(* Logix 5000 project; controller Evlog vendor 1 type 14 code 15 rev 20.11; software revision 20.05 *)

TASK MainTask (continuous, watchdog 500 ms) : MainProgram

MODULES
   Local : vendor 1 type 14 code 15 (SoftLogixController 2, rev 20.11)
      EIP : vendor 1 type 12 code 135 (SoftLogixVB 3, Ethernet 172.22.255.153, rev 20.1)
END_MODULES

TYPE STRING484 :
STRUCT
   LEN : DINT;
   DATA : SINT[480];
END_STRUCT
END_TYPE

TYPE u_EventTable :
STRUCT
   Ons_Short : BOOL[512];
   Last_Status : BOOL[1024];
END_STRUCT
END_TYPE

TYPE u_Timer :
STRUCT
   Yer : INT;
   Month : SINT;
   Day : SINT;
   Hour : SINT;
   Minute : SINT;
   Sec : SINT;
   MillSec : DINT;
END_STRUCT
END_TYPE

TYPE uEventsDB :
STRUCT
   Events : uEvlent[1024];
   NextEvent : INT;
   LastLostEvent : INT;
   EventOverFlow : BOOL;
   RemainderValidEvent : INT;
END_STRUCT
END_TYPE

TYPE uEvlent :   // @Ver 1.0
STRUCT
   ID : INT;   // Event ID
   Active : BOOL;
   IsSend : BOOL;
   Time : u_Timer;
END_STRUCT
END_TYPE

TYPE uSendMsg :   // @Ver 1.0
STRUCT
   MsgCount : SINT;
   BufferNotEmpty : BOOL;
   EmptyBuffer : uEvlent;
   SendBuffer : uEvlent;
   SendMSG : STRING;
END_STRUCT
END_TYPE

ADD_ON_INSTRUCTION CreateSendEvent   (* revision 1.0 *)
VAR_IN_OUT
   io_EvDB : uEventsDB; {required}
   o_SendBuffer : uSendMsg; {required}
END_VAR
VAR_INPUT
   Mutil_EvSend : BOOL; {access None, visible}
END_VAR
VAR_OUTPUT
   o_Error : BOOL; {access None}
END_VAR
VAR
   LocalEvDB : uEventsDB; {access None}
   True : BOOL; {access None}
   False : BOOL; {access None}
   i : DINT; {access None}
   Max_MsgCount : DINT; {access None}
   Last_index : DINT; {access None}
   MsgIndex : DINT; {access None}
   Temp_ID : STRING; {access None}
   Temp_Time : STRING; {access None}
   TIMEToSTRING : TIME_To_STRING; {access None}
   Index : DINT; {access None}
   Delimit : SINT; {access None}
   Split : STRING; {access None}
   Temp_Str : STRING; {access None}
   Time2Str : TIME_To_STRING; {access None}
   tempCount : DINT; {access None}
   EndOfCount : DINT; {access None}
   Tem_Str1 : STRING; {access None}
END_VAR

ROUTINE Logic   (* structured text *)
   
   True :=1;
   False:=0;
   Split.DATA[0]:=58;
   Split.Len:=1;
   Max_MsgCount:=500;
   o_Error:=False;
   Temp_Str.Len:=0;
   
   //
   
   IF Not o_SendBuffer.BufferNotEmpty Then
      o_SendBuffer.SendMSG.Len:=0;
   END_IF;
   
   //Mssage: ID:Timer:
   IF  io_EvDB.NextEvent>1 AND Not o_SendBuffer.BufferNotEmpty Then
       IF Not Mutil_EvSend then
   	   Cop(io_EvDB.Events[io_EvDB.NextEvent-1], o_SendBuffer.SendBuffer,1);
          //Cop(o_SendBuffer.EmptyBuffer, io_EvDB.Events[io_EvDB.NextEvent],1);
          DTOS(o_SendBuffer.SendBuffer.ID,Temp_Str);
   	   Concat(o_SendBuffer.SendMSG,Temp_Str,o_SendBuffer.SendMSG);
   	   Temp_Str.Len:=0;
          Concat(o_SendBuffer.SendMSG,Split,o_SendBuffer.SendMSG);
          TIME_To_STRING(Time2Str,o_SendBuffer.SendBuffer.Time,Temp_Str);
   	   Concat(o_SendBuffer.SendMSG,Temp_Str,o_SendBuffer.SendMSG);
          o_SendBuffer.BufferNotEmpty:=True;
          io_EvDB.NextEvent:=io_EvDB.NextEvent-1;
   	END_IF;
   
   END_IF;
   
   
   
   
   
   
   
   
   
   
   
   
   
   
   
   
   
   
   
   
   
   
   
   
   
   
   
   
   
   
   
   
   
   
   
   
   
   
   
   
   
   
   
   
   
   
   
END_ROUTINE
END_ADD_ON_INSTRUCTION

ADD_ON_INSTRUCTION CreatNewEvent   (* revision 1.0 *)
VAR_INPUT
   Enbale : DINT;
   Single_Input : BOOL; {required}
   Ev_ID : DINT; {access None, required}
END_VAR
VAR_IN_OUT
   IO_EvDB : uEventsDB; {required}
END_VAR
VAR_INPUT
   o_Parem_Err : BOOL; {access None, required}
END_VAR
VAR_IN_OUT
   Ev_Table : u_EventTable; {required}
END_VAR
VAR
   DT : DINT[6]; {access None}
   LocalIndex : DINT; {access None}
   Single_Trig : BOOL[1024]; {access None}
   OnsHelper : BOOL[1024]; {access None}
   Temp_SwitchSingle : BOOL; {access None}
   False : BOOL; {access None}
   True : BOOL; {access None}
   Max_ID : DINT; {access None}
   LocalDateTime : DINT[7]; {access None}
   Local_EvDB : uEvlent[1001]; {access None}
END_VAR

ROUTINE Logic   (* structured text *)
   
   (*
   VERSIONS:
   
   V1.0    |   Jerry  | First release
   
   
   1.单周期内  如果ID不一致 ,产生新的事件记录
   2.不同周期下,如果信号被重新触发,产生新的事件记录.
   3.同一事件,如果下一个周期没有产生上升沿 将不会记录.
   
   *)
   
   (*
   VERSION : '1.0'
   AUTHOR  : Jerry
   NAME    : EVENT
   FAMILY  : global
   *)
   
   True   :=1;
   False  :=0;
   Max_ID :=1000;//此处UDT 定义为1024
   
   Temp_SwitchSingle:=Single_Input;    //Cop  到本地 确保  本次程序结束能够复位状态,使下一次调用重新初始化
   IF Ev_ID>Max_ID OR Ev_ID<=0 Then
      o_Parem_Err:=True;
      Ev_ID:=1;
   END_IF;
   
   IF IO_EvDB.NextEvent>Max_ID OR IO_EvDB.NextEvent<=0 Then
      IO_EvDB.NextEvent:=1;
   END_IF;
   
   IF  Temp_SwitchSingle and not Ev_Table.Last_Status[Ev_ID] then
       Ev_Table.Last_Status[Ev_ID]:=True;
   //添加事件时间到Buffer
       GSV(WallClockTime,,DateTime,LocalDateTime[0]);
       IO_EvDB.Events[IO_EvDB.NextEvent].Time.Yer   :=LocalDateTime[0];
       IO_EvDB.Events[IO_EvDB.NextEvent].Time.Month :=LocalDateTime[1];
   	IO_EvDB.Events[IO_EvDB.NextEvent].Time.day   :=LocalDateTime[2];
   	IO_EvDB.Events[IO_EvDB.NextEvent].Time.hour  :=LocalDateTime[3];
   	IO_EvDB.Events[IO_EvDB.NextEvent].Time.minute:=LocalDateTime[4];
   	IO_EvDB.Events[IO_EvDB.NextEvent].Time.Sec   :=LocalDateTime[5];
   	IO_EvDB.Events[IO_EvDB.NextEvent].Time.MillSec:=LocalDateTime[6];
   
   	//添加事件ID到Buffer
   	IO_EvDB.Events[IO_EvDB.NextEvent].ID:=Ev_ID;
   	IO_EvDB.Events[IO_EvDB.NextEvent].Active:=True;
       IO_EvDB.Events[IO_EvDB.NextEvent].IsSend:=False;
   	IO_EvDB.NextEvent:=IO_EvDB.NextEvent+1;
   	IO_EvDB.RemainderValidEvent:=IO_EvDB.RemainderValidEvent+1;
   	IF IO_EvDB.NextEvent>Max_ID then
   	   IO_EvDB.NextEvent:=1;
          IO_EvDB.EventOverFlow:=True;
   	END_IF;
   End_IF;
   
   
   IF Not Temp_SwitchSingle and Ev_Table.Last_Status[Ev_ID] then
      Ev_Table.Last_Status[Ev_ID]:=False;
   END_IF;
   
   
   
   
   
END_ROUTINE
END_ADD_ON_INSTRUCTION

ADD_ON_INSTRUCTION CreatSendMsg   (* revision 1.0 *)
VAR_IN_OUT
   io_EvDB : uEventsDB; {required}
   o_SendMSG : uSendMsg; {required}
   Time2Str1 : TIME_To_STRING; {required}
END_VAR
VAR
   Split : STRING := ':'; {access None}
   Temp_Str : STRING; {access None}
   Time2Str : TIME_To_STRING; {access None}
END_VAR

ROUTINE Logic   (* ladder *)
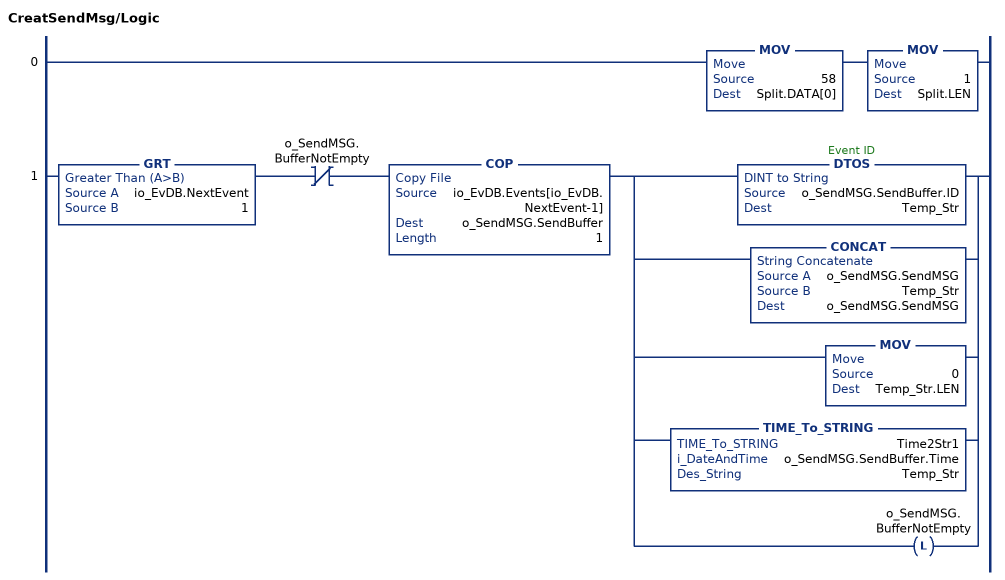
   0: MOV(58,Split.DATA[0])MOV(1,Split.LEN);
   1: GRT(io_EvDB.NextEvent,1)XIO(o_SendMSG.BufferNotEmpty)COP(io_EvDB.Events[io_EvDB.NextEvent-1],o_SendMSG.SendBuffer,1)[DTOS(o_SendMSG.SendBuffer.ID,Temp_Str) ,CONCAT(o_SendMSG.SendMSG,Temp_Str,o_SendMSG.SendMSG) ,MOV(0,Temp_Str.LEN) ,TIME_To_STRING(Time2Str1,o_SendMSG.SendBuffer.Time,Temp_Str) ,OTL(o_SendMSG.BufferNotEmpty) ];
END_ROUTINE
END_ADD_ON_INSTRUCTION

ADD_ON_INSTRUCTION TIME_To_STRING   (* revision 1.0 *)
VAR_IN_OUT
   i_DateAndTime : u_Timer; {required}
   Des_String : STRING; {required}
END_VAR
VAR
   i : DINT; {access None}
   Temp_Str : STRING; {access None}
   Split : STRING := '.'; {access None}
END_VAR

ROUTINE Logic   (* structured text *)
   
   
   Des_String.len:=0;
         DTOS(i_DateAndTime.Yer,Temp_Str);
      Concat(Des_String,Temp_Str,Des_String);
      Concat(Des_String,Split,Des_String);
      Temp_Str.Len:=0;
         DTOS(i_DateAndTime.Month,Temp_Str);
      Concat(Des_String,Temp_Str,Des_String);
      Concat(Des_String,Split,Des_String);
      Temp_Str.Len:=0;
         DTOS(i_DateAndTime.Day,Temp_Str);
      Concat(Des_String,Temp_Str,Des_String);
      Concat(Des_String,Split,Des_String);
      Temp_Str.Len:=0;
         DTOS(i_DateAndTime.Hour,Temp_Str);
      Concat(Des_String,Temp_Str,Des_String);
      Concat(Des_String,Split,Des_String);
      Temp_Str.Len:=0;
         DTOS(i_DateAndTime.Minute,Temp_Str);
      Concat(Des_String,Temp_Str,Des_String);
      Concat(Des_String,Split,Des_String);
      Temp_Str.Len:=0;
          DTOS(i_DateAndTime.Sec,Temp_Str);
      Concat(Des_String,Temp_Str,Des_String);
      Concat(Des_String,Split,Des_String);
   Temp_Str.Len:=0;
          DTOS(i_DateAndTime.MillSec,Temp_Str);
      Concat(Des_String,Temp_Str,Des_String);
END_ROUTINE
END_ADD_ON_INSTRUCTION

VAR_GLOBAL   (* controller tags *)
   booltest : BOOL := 1;
   Ev_Table : u_EventTable;
   EvMsgDB : uEvlent[10000];
   SendBuffer : uSendMsg := (MsgCount := 1, SendBuffer.ID := 1, SendBuffer.Active := 1, SendBuffer.Time.Yer := 2022, SendBuffer.Time.Month := 2, SendBuffer.Time.Day := 5, SendBuffer.Time.Hour := 14, SendBuffer.Time.Minute := 40, SendBuffer.Time.Sec := 40, SendBuffer.Time.MillSec := 175138);
   SendMsg_Buffer : uSendMsg := (BufferNotEmpty := 1);
   string1 : STRING := '123456';
   test : BOOL;
   testStr : STRING;
   Time2Str : TIME_To_STRING;
END_VAR

PROGRAM MainProgram   (* main routine MainRoutine *)
VAR
   CreatMSG : CreatSendMsg;
   ddd : DINT := 2022;
   Ev_Table : u_EventTable := (Last_Status[1] := 1);
   EvDB : uEvlent[1000] := ([0].ID := 1, [0].Active := 1, [1].ID := 2, [1].Active := 1, [2].ID := 1, [2].Active := 1, [3].ID := 2, [3].Active := 1, [4].ID := 1, [4].Active := 1, [5].ID := 2, [5].Active := 1, [6].ID := 1, [6].Active := 1, [7].ID := 2, [7].Active := 1, [8].ID := 1, [8].Active := 1, [9].ID := 2, [9].Active := 1, [10].ID := 1, [10].Active := 1, [11].ID := 2, [11].Active := 1, [12].ID := 1, [12].Active := 1, [13].ID := 2, [13].Active := 1, [14].ID := 1, [14].Active := 1, [15].ID := 2, [15].Active := 1, [16].ID := 1, [16].Active := 1, [17].ID := 2, [17].Active := 1, [18].ID := 1, [18].Active := 1, [19].ID := 2, [19].Active := 1, [20].ID := 1, [20].Active := 1, [21].ID := 2, [21].Active := 1, [22].ID := 1, [22].Active := 1, [23].ID := 2, [23].Active := 1, [24].ID := 1, [24].Active := 1, [25].ID := 2, [25].Active := 1, [26].ID := 1, [26].Active := 1, [27].ID := 2, [27].Active := 1, [28].ID := 1, [28].Active := 1, [29].ID := 2, [29].Active := 1,
        [30].ID := 1, [30].Active := 1, [31].ID := 2, [31].Active := 1, [32].ID := 1, [32].Active := 1, [33].ID := 2, [33].Active := 1, [34].ID := 1, [34].Active := 1, [35].ID := 2, [35].Active := 1, [36].ID := 1, [36].Active := 1, [37].ID := 2, [37].Active := 1, [38].ID := 1, [38].Active := 1, [39].ID := 2, [39].Active := 1, [40].ID := 1, [40].Active := 1, [41].ID := 2, [41].Active := 1, [42].ID := 1, [42].Active := 1, [43].ID := 2, [43].Active := 1, [44].ID := 1, [44].Active := 1, [45].ID := 2, [45].Active := 1, [46].ID := 1, [46].Active := 1, [47].ID := 2, [47].Active := 1, [48].ID := 1, [48].Active := 1, [49].ID := 2, [49].Active := 1, [50].ID := 1, [50].Active := 1, [51].ID := 2, [51].Active := 1, [52].ID := 1, [52].Active := 1, [53].ID := 2, [53].Active := 1, [54].ID := 1, [54].Active := 1, [55].ID := 2, [55].Active := 1, [56].ID := 1, [56].Active := 1, [57].ID := 2, [57].Active := 1, [58].ID := 1, [58].Active := 1, [59].ID := 2, [59].Active := 1,
        [60].ID := 1, [60].Active := 1, [61].ID := 2, [61].Active := 1, [62].ID := 1, [62].Active := 1, [63].ID := 2, [63].Active := 1, [64].ID := 1, [64].Active := 1, [65].ID := 2, [65].Active := 1, [66].ID := 1, [66].Active := 1, [67].ID := 2, [67].Active := 1, [68].ID := 1, [68].Active := 1, [69].ID := 2, [69].Active := 1, [70].ID := 1, [70].Active := 1, [71].ID := 2, [71].Active := 1, [72].ID := 1, [72].Active := 1, [73].ID := 2, [73].Active := 1, [74].ID := 1, [74].Active := 1, [75].ID := 2, [75].Active := 1, [76].ID := 1, [76].Active := 1, [77].ID := 2, [77].Active := 1, [78].ID := 1, [78].Active := 1, [79].ID := 2, [79].Active := 1, [80].ID := 1, [80].Active := 1, [81].ID := 2, [81].Active := 1, [82].ID := 1, [82].Active := 1, [83].ID := 2, [83].Active := 1, [84].ID := 1, [84].Active := 1, [85].ID := 2, [85].Active := 1, [86].ID := 1, [86].Active := 1, [87].ID := 2, [87].Active := 1, [88].ID := 1, [88].Active := 1, [89].ID := 2, [89].Active := 1,
        [90].ID := 1, [90].Active := 1, [91].ID := 2, [91].Active := 1, [92].ID := 1, [92].Active := 1, [93].ID := 2, [93].Active := 1, [94].ID := 1, [94].Active := 1, [95].ID := 2, [95].Active := 1, [96].ID := 1, [96].Active := 1, [97].ID := 2, [97].Active := 1, [98].ID := 1, [98].Active := 1, [99].ID := 2, [99].Active := 1, [100].ID := 1, [100].Active := 1, [101].ID := 2, [101].Active := 1, [102].ID := 1, [102].Active := 1, [103].ID := 2, [103].Active := 1, [104].ID := 1, [104].Active := 1, [105].ID := 2, [105].Active := 1, [106].ID := 1, [106].Active := 1, [107].ID := 2, [107].Active := 1, [108].ID := 1, [108].Active := 1, [109].ID := 2, [109].Active := 1, [110].ID := 1, [110].Active := 1, [111].ID := 2, [111].Active := 1, [112].ID := 1, [112].Active := 1, [113].ID := 2, [113].Active := 1, [114].ID := 1, [114].Active := 1, [115].ID := 2, [115].Active := 1, [116].ID := 1, [116].Active := 1, [117].ID := 2, [117].Active := 1, [118].ID := 1, [118].Active := 1, [119].ID := 2, [119].Active := 1,
        [120].ID := 1, [120].Active := 1, [121].ID := 2, [121].Active := 1, [122].ID := 1, [122].Active := 1, [123].ID := 2, [123].Active := 1, [124].ID := 1, [124].Active := 1, [125].ID := 2, [125].Active := 1, [126].ID := 1, [126].Active := 1, [127].ID := 2, [127].Active := 1, [128].ID := 1, [128].Active := 1, [129].ID := 2, [129].Active := 1, [130].ID := 1, [130].Active := 1, [131].ID := 2, [131].Active := 1, [132].ID := 1, [132].Active := 1, [133].ID := 2, [133].Active := 1, [134].ID := 1, [134].Active := 1, [135].ID := 2, [135].Active := 1, [136].ID := 1, [136].Active := 1, [137].ID := 2, [137].Active := 1, [138].ID := 1, [138].Active := 1, [139].ID := 2, [139].Active := 1, [140].ID := 1, [140].Active := 1, [141].ID := 2, [141].Active := 1, [142].ID := 1, [142].Active := 1, [143].ID := 2, [143].Active := 1, [144].ID := 1, [144].Active := 1, [145].ID := 2, [145].Active := 1, [146].ID := 1, [146].Active := 1, [147].ID := 2, [147].Active := 1, [148].ID := 1, [148].Active := 1, [149].ID := 2, [149].Active := 1,
        [150].ID := 1, [150].Active := 1, [151].ID := 2, [151].Active := 1, [152].ID := 1, [152].Active := 1, [153].ID := 2, [153].Active := 1, [154].ID := 1, [154].Active := 1, [155].ID := 2, [155].Active := 1, [156].ID := 1, [156].Active := 1, [157].ID := 2, [157].Active := 1, [158].ID := 1, [158].Active := 1, [159].ID := 2, [159].Active := 1, [160].ID := 1, [160].Active := 1, [161].ID := 2, [161].Active := 1, [162].ID := 1, [162].Active := 1, [163].ID := 2, [163].Active := 1, [164].ID := 1, [164].Active := 1, [165].ID := 2, [165].Active := 1, [166].ID := 1, [166].Active := 1, [167].ID := 2, [167].Active := 1, [168].ID := 1, [168].Active := 1, [169].ID := 2, [169].Active := 1, [170].ID := 1, [170].Active := 1, [171].ID := 2, [171].Active := 1, [172].ID := 2, [172].Active := 1, [173].ID := 1, [173].Active := 1, [174].ID := 2, [174].Active := 1, [175].ID := 1, [175].Active := 1, [176].ID := 2, [176].Active := 1, [177].ID := 1, [177].Active := 1, [178].ID := 2, [178].Active := 1, [179].ID := 1, [179].Active := 1,
        [180].ID := 2, [180].Active := 1, [181].ID := 1, [181].Active := 1, [182].ID := 2, [182].Active := 1, [183].ID := 1, [183].Active := 1, [184].ID := 2, [184].Active := 1, [185].ID := 1, [185].Active := 1, [186].ID := 2, [186].Active := 1, [187].ID := 1, [187].Active := 1, [188].ID := 2, [188].Active := 1, [189].ID := 1, [189].Active := 1, [190].ID := 2, [190].Active := 1, [191].ID := 1, [191].Active := 1, [192].ID := 2, [192].Active := 1, [193].ID := 1, [193].Active := 1, [194].ID := 2, [194].Active := 1, [195].ID := 1, [195].Active := 1, [196].ID := 2, [196].Active := 1, [197].ID := 1, [197].Active := 1, [198].ID := 2, [198].Active := 1, [199].ID := 1, [199].Active := 1, [200].ID := 2, [200].Active := 1, [201].ID := 1, [201].Active := 1, [202].ID := 2, [202].Active := 1, [203].ID := 1, [203].Active := 1, [204].ID := 2, [204].Active := 1, [205].ID := 1, [205].Active := 1, [206].ID := 2, [206].Active := 1, [207].ID := 1, [207].Active := 1, [208].ID := 2, [208].Active := 1, [209].ID := 1, [209].Active := 1,
        [210].ID := 2, [210].Active := 1, [211].ID := 1, [211].Active := 1, [212].ID := 2, [212].Active := 1, [213].ID := 1, [213].Active := 1, [214].ID := 2, [214].Active := 1, [215].ID := 1, [215].Active := 1, [216].ID := 2, [216].Active := 1, [217].ID := 1, [217].Active := 1, [218].ID := 2, [218].Active := 1, [219].ID := 1, [219].Active := 1, [220].ID := 2, [220].Active := 1, [221].ID := 1, [221].Active := 1, [222].ID := 2, [222].Active := 1, [223].ID := 1, [223].Active := 1, [224].ID := 2, [224].Active := 1, [225].ID := 1, [225].Active := 1, [226].ID := 2, [226].Active := 1, [227].ID := 1, [227].Active := 1, [228].ID := 2, [228].Active := 1, [229].ID := 1, [229].Active := 1, [230].ID := 2, [230].Active := 1, [231].ID := 1, [231].Active := 1, [232].ID := 2, [232].Active := 1, [233].ID := 1, [233].Active := 1, [234].ID := 2, [234].Active := 1, [235].ID := 1, [235].Active := 1, [236].ID := 2, [236].Active := 1, [237].ID := 1, [237].Active := 1, [238].ID := 2, [238].Active := 1, [239].ID := 1, [239].Active := 1,
        [240].ID := 2, [240].Active := 1, [241].ID := 1, [241].Active := 1, [242].ID := 2, [242].Active := 1, [243].ID := 1, [243].Active := 1, [244].ID := 2, [244].Active := 1, [245].ID := 1, [245].Active := 1, [246].ID := 2, [246].Active := 1, [247].ID := 1, [247].Active := 1, [248].ID := 2, [248].Active := 1, [249].ID := 1, [249].Active := 1, [250].ID := 2, [250].Active := 1, [251].ID := 1, [251].Active := 1, [252].ID := 2, [252].Active := 1, [253].ID := 1, [253].Active := 1, [254].ID := 2, [254].Active := 1, [255].ID := 1, [255].Active := 1, [256].ID := 2, [256].Active := 1, [257].ID := 1, [257].Active := 1, [258].ID := 2, [258].Active := 1, [259].ID := 1, [259].Active := 1, [260].ID := 2, [260].Active := 1, [261].ID := 1, [261].Active := 1, [262].ID := 2, [262].Active := 1, [263].ID := 1, [263].Active := 1, [264].ID := 2, [264].Active := 1, [265].ID := 1, [265].Active := 1, [266].ID := 2, [266].Active := 1, [267].ID := 1, [267].Active := 1, [268].ID := 2, [268].Active := 1, [269].ID := 1, [269].Active := 1,
        [270].ID := 2, [270].Active := 1, [271].ID := 1, [271].Active := 1, [272].ID := 2, [272].Active := 1, [273].ID := 1, [273].Active := 1, [274].ID := 2, [274].Active := 1, [275].ID := 1, [275].Active := 1, [276].ID := 2, [276].Active := 1, [277].ID := 1, [277].Active := 1, [278].ID := 2, [278].Active := 1, [279].ID := 1, [279].Active := 1, [280].ID := 2, [280].Active := 1, [281].ID := 1, [281].Active := 1, [282].ID := 2, [282].Active := 1, [283].ID := 1, [283].Active := 1, [284].ID := 2, [284].Active := 1, [285].ID := 1, [285].Active := 1, [286].ID := 2, [286].Active := 1, [287].ID := 1, [287].Active := 1, [288].ID := 2, [288].Active := 1, [289].ID := 1, [289].Active := 1, [290].ID := 2, [290].Active := 1, [291].ID := 1, [291].Active := 1, [292].ID := 2, [292].Active := 1, [293].ID := 1, [293].Active := 1, [294].ID := 2, [294].Active := 1, [295].ID := 1, [295].Active := 1, [296].ID := 2, [296].Active := 1, [297].ID := 1, [297].Active := 1, [298].ID := 2, [298].Active := 1, [299].ID := 1, [299].Active := 1,
        [300].ID := 2, [300].Active := 1, [301].ID := 1, [301].Active := 1, [302].ID := 2, [302].Active := 1, [303].ID := 1, [303].Active := 1, [304].ID := 2, [304].Active := 1, [305].ID := 1, [305].Active := 1, [306].ID := 2, [306].Active := 1, [307].ID := 1, [307].Active := 1, [308].ID := 2, [308].Active := 1, [309].ID := 1, [309].Active := 1, [310].ID := 2, [310].Active := 1, [311].ID := 1, [311].Active := 1, [312].ID := 2, [312].Active := 1, [313].ID := 1, [313].Active := 1, [314].ID := 2, [314].Active := 1, [315].ID := 1, [315].Active := 1, [316].ID := 2, [316].Active := 1, [317].ID := 1, [317].Active := 1, [318].ID := 2, [318].Active := 1, [319].ID := 1, [319].Active := 1, [320].ID := 2, [320].Active := 1, [321].ID := 1, [321].Active := 1, [322].ID := 2, [322].Active := 1, [323].ID := 1, [323].Active := 1, [324].ID := 2, [324].Active := 1, [325].ID := 1, [325].Active := 1, [326].ID := 2, [326].Active := 1, [327].ID := 1, [327].Active := 1, [328].ID := 2, [328].Active := 1, [329].ID := 1, [329].Active := 1,
        [330].ID := 2, [330].Active := 1, [331].ID := 1, [331].Active := 1, [332].ID := 2, [332].Active := 1, [333].ID := 1, [333].Active := 1, [334].ID := 2, [334].Active := 1, [335].ID := 1, [335].Active := 1, [336].ID := 2, [336].Active := 1, [337].ID := 1, [337].Active := 1, [338].ID := 2, [338].Active := 1, [339].ID := 1, [339].Active := 1, [340].ID := 2, [340].Active := 1, [341].ID := 1, [341].Active := 1, [342].ID := 2, [342].Active := 1, [343].ID := 1, [343].Active := 1, [344].ID := 2, [344].Active := 1, [345].ID := 1, [345].Active := 1, [346].ID := 2, [346].Active := 1, [347].ID := 1, [347].Active := 1, [348].ID := 2, [348].Active := 1, [349].ID := 1, [349].Active := 1, [350].ID := 2, [350].Active := 1, [351].ID := 1, [351].Active := 1, [352].ID := 2, [352].Active := 1, [353].ID := 1, [353].Active := 1, [354].ID := 2, [354].Active := 1, [355].ID := 1, [355].Active := 1, [356].ID := 2, [356].Active := 1, [357].ID := 1, [357].Active := 1, [358].ID := 2, [358].Active := 1, [359].ID := 1, [359].Active := 1,
        [360].ID := 2, [360].Active := 1, [361].ID := 1, [361].Active := 1, [362].ID := 2, [362].Active := 1, [363].ID := 1, [363].Active := 1, [364].ID := 2, [364].Active := 1, [365].ID := 1, [365].Active := 1, [366].ID := 2, [366].Active := 1, [367].ID := 1, [367].Active := 1, [368].ID := 2, [368].Active := 1, [369].ID := 1, [369].Active := 1, [370].ID := 2, [370].Active := 1, [371].ID := 1, [371].Active := 1, [372].ID := 2, [372].Active := 1, [373].ID := 1, [373].Active := 1, [374].ID := 2, [374].Active := 1, [375].ID := 1, [375].Active := 1, [376].ID := 2, [376].Active := 1, [377].ID := 1, [377].Active := 1, [378].ID := 2, [378].Active := 1, [379].ID := 1, [379].Active := 1, [380].ID := 2, [380].Active := 1, [381].ID := 1, [381].Active := 1, [382].ID := 2, [382].Active := 1, [383].ID := 1, [383].Active := 1, [384].ID := 2, [384].Active := 1, [385].ID := 1, [385].Active := 1, [386].ID := 2, [386].Active := 1, [387].ID := 1, [387].Active := 1, [388].ID := 2, [388].Active := 1, [389].ID := 1, [389].Active := 1,
        [390].ID := 2, [390].Active := 1, [391].ID := 1, [391].Active := 1, [392].ID := 2, [392].Active := 1, [393].ID := 1, [393].Active := 1, [394].ID := 2, [394].Active := 1, [395].ID := 1, [395].Active := 1, [396].ID := 2, [396].Active := 1, [397].ID := 1, [397].Active := 1, [398].ID := 2, [398].Active := 1, [399].ID := 1, [399].Active := 1, [400].ID := 2, [400].Active := 1, [401].ID := 1, [401].Active := 1, [402].ID := 2, [402].Active := 1, [403].ID := 1, [403].Active := 1, [404].ID := 2, [404].Active := 1, [405].ID := 1, [405].Active := 1, [406].ID := 2, [406].Active := 1, [407].ID := 1, [407].Active := 1, [408].ID := 2, [408].Active := 1, [409].ID := 1, [409].Active := 1, [410].ID := 2, [410].Active := 1, [411].ID := 1, [411].Active := 1, [412].ID := 2, [412].Active := 1, [413].ID := 1, [413].Active := 1, [414].ID := 2, [414].Active := 1, [415].ID := 1, [415].Active := 1, [416].ID := 2, [416].Active := 1, [417].ID := 1, [417].Active := 1, [418].ID := 2, [418].Active := 1, [419].ID := 1, [419].Active := 1,
        [420].ID := 2, [420].Active := 1, [421].ID := 1, [421].Active := 1, [422].ID := 2, [422].Active := 1, [423].ID := 1, [423].Active := 1, [424].ID := 2, [424].Active := 1, [425].ID := 1, [425].Active := 1, [426].ID := 2, [426].Active := 1, [427].ID := 1, [427].Active := 1, [428].ID := 2, [428].Active := 1, [429].ID := 1, [429].Active := 1, [430].ID := 2, [430].Active := 1, [431].ID := 1, [431].Active := 1, [432].ID := 2, [432].Active := 1, [433].ID := 1, [433].Active := 1, [434].ID := 2, [434].Active := 1, [435].ID := 1, [435].Active := 1, [436].ID := 2, [436].Active := 1, [437].ID := 1, [437].Active := 1, [438].ID := 2, [438].Active := 1, [439].ID := 1, [439].Active := 1, [440].ID := 2, [440].Active := 1, [441].ID := 1, [441].Active := 1, [442].ID := 2, [442].Active := 1, [443].ID := 1, [443].Active := 1, [444].ID := 2, [444].Active := 1, [445].ID := 1, [445].Active := 1, [446].ID := 2, [446].Active := 1, [447].ID := 1, [447].Active := 1, [448].ID := 2, [448].Active := 1, [449].ID := 1, [449].Active := 1,
        [450].ID := 2, [450].Active := 1, [451].ID := 1, [451].Active := 1, [452].ID := 2, [452].Active := 1, [453].ID := 1, [453].Active := 1, [454].ID := 2, [454].Active := 1, [455].ID := 1, [455].Active := 1, [456].ID := 2, [456].Active := 1, [457].ID := 1, [457].Active := 1, [458].ID := 2, [458].Active := 1, [459].ID := 1, [459].Active := 1, [460].ID := 2, [460].Active := 1, [461].ID := 1, [461].Active := 1, [462].ID := 2, [462].Active := 1, [463].ID := 1, [463].Active := 1, [464].ID := 2, [464].Active := 1, [465].ID := 1, [465].Active := 1, [466].ID := 2, [466].Active := 1, [467].ID := 1, [467].Active := 1, [468].ID := 2, [468].Active := 1, [469].ID := 1, [469].Active := 1, [470].ID := 2, [470].Active := 1, [471].ID := 1, [471].Active := 1, [472].ID := 2, [472].Active := 1, [473].ID := 1, [473].Active := 1, [474].ID := 2, [474].Active := 1, [475].ID := 1, [475].Active := 1, [476].ID := 2, [476].Active := 1, [477].ID := 1, [477].Active := 1, [478].ID := 2, [478].Active := 1, [479].ID := 1, [479].Active := 1,
        [480].ID := 2, [480].Active := 1, [481].ID := 1, [481].Active := 1, [482].ID := 2, [482].Active := 1, [483].ID := 1, [483].Active := 1, [484].ID := 2, [484].Active := 1, [485].ID := 1, [485].Active := 1, [486].ID := 2, [486].Active := 1, [487].ID := 1, [487].Active := 1, [488].ID := 2, [488].Active := 1, [489].ID := 1, [489].Active := 1, [490].ID := 2, [490].Active := 1, [491].ID := 1, [491].Active := 1, [492].ID := 2, [492].Active := 1, [493].ID := 1, [493].Active := 1, [494].ID := 2, [494].Active := 1, [495].ID := 1, [495].Active := 1, [496].ID := 2, [496].Active := 1, [497].ID := 1, [497].Active := 1, [498].ID := 2, [498].Active := 1, [499].ID := 1, [499].Active := 1, [500].ID := 2, [500].Active := 1, [501].ID := 1, [501].Active := 1, [502].ID := 2, [502].Active := 1, [503].ID := 1, [503].Active := 1, [504].ID := 2, [504].Active := 1, [505].ID := 1, [505].Active := 1, [506].ID := 2, [506].Active := 1, [507].ID := 1, [507].Active := 1, [508].ID := 2, [508].Active := 1, [509].ID := 1, [509].Active := 1,
        [510].ID := 2, [510].Active := 1, [511].ID := 1, [511].Active := 1, [512].ID := 2, [512].Active := 1, [513].ID := 1, [513].Active := 1, [514].ID := 2, [514].Active := 1, [515].ID := 1, [515].Active := 1, [516].ID := 2, [516].Active := 1, [517].ID := 1, [517].Active := 1, [518].ID := 2, [518].Active := 1, [519].ID := 1, [519].Active := 1, [520].ID := 2, [520].Active := 1, [521].ID := 1, [521].Active := 1, [522].ID := 2, [522].Active := 1, [523].ID := 1, [523].Active := 1, [524].ID := 2, [524].Active := 1, [525].ID := 1, [525].Active := 1, [526].ID := 2, [526].Active := 1, [527].ID := 1, [527].Active := 1, [528].ID := 2, [528].Active := 1, [529].ID := 1, [529].Active := 1, [530].ID := 2, [530].Active := 1, [531].ID := 1, [531].Active := 1, [532].ID := 2, [532].Active := 1, [533].ID := 1, [533].Active := 1, [534].ID := 2, [534].Active := 1, [535].ID := 1, [535].Active := 1, [536].ID := 2, [536].Active := 1, [537].ID := 1, [537].Active := 1, [538].ID := 2, [538].Active := 1, [539].ID := 1, [539].Active := 1,
        [540].ID := 2, [540].Active := 1, [541].ID := 1, [541].Active := 1, [542].ID := 2, [542].Active := 1, [543].ID := 1, [543].Active := 1, [544].ID := 2, [544].Active := 1, [545].ID := 1, [545].Active := 1, [546].ID := 2, [546].Active := 1, [547].ID := 1, [547].Active := 1, [548].ID := 2, [548].Active := 1, [549].ID := 1, [549].Active := 1, [550].ID := 2, [550].Active := 1, [551].ID := 1, [551].Active := 1, [552].ID := 2, [552].Active := 1, [553].ID := 1, [553].Active := 1, [554].ID := 2, [554].Active := 1, [555].ID := 1, [555].Active := 1, [556].ID := 2, [556].Active := 1, [557].ID := 1, [557].Active := 1, [558].ID := 2, [558].Active := 1, [559].ID := 1, [559].Active := 1, [560].ID := 2, [560].Active := 1, [561].ID := 1, [561].Active := 1, [562].ID := 2, [562].Active := 1, [563].ID := 1, [563].Active := 1, [564].ID := 2, [564].Active := 1, [565].ID := 1, [565].Active := 1, [566].ID := 2, [566].Active := 1, [567].ID := 1, [567].Active := 1, [568].ID := 2, [568].Active := 1, [569].ID := 1, [569].Active := 1,
        [570].ID := 2, [570].Active := 1, [571].ID := 1, [571].Active := 1, [572].ID := 2, [572].Active := 1, [573].ID := 1, [573].Active := 1, [574].ID := 2, [574].Active := 1, [575].ID := 1, [575].Active := 1, [576].ID := 2, [576].Active := 1, [577].ID := 1, [577].Active := 1, [578].ID := 2, [578].Active := 1, [579].ID := 1, [579].Active := 1, [580].ID := 2, [580].Active := 1, [581].ID := 1, [581].Active := 1, [582].ID := 2, [582].Active := 1, [583].ID := 1, [583].Active := 1, [584].ID := 2, [584].Active := 1, [585].ID := 1, [585].Active := 1, [586].ID := 2, [586].Active := 1, [587].ID := 1, [587].Active := 1, [588].ID := 2, [588].Active := 1, [589].ID := 1, [589].Active := 1, [590].ID := 2, [590].Active := 1, [591].ID := 1, [591].Active := 1, [592].ID := 2, [592].Active := 1, [593].ID := 1, [593].Active := 1, [594].ID := 2, [594].Active := 1, [595].ID := 1, [595].Active := 1, [596].ID := 2, [596].Active := 1, [597].ID := 1, [597].Active := 1, [598].ID := 2, [598].Active := 1, [599].ID := 1, [599].Active := 1,
        [600].ID := 2, [600].Active := 1, [601].ID := 1, [601].Active := 1, [602].ID := 2, [602].Active := 1, [603].ID := 1, [603].Active := 1, [604].ID := 2, [604].Active := 1, [605].ID := 1, [605].Active := 1, [606].ID := 2, [606].Active := 1, [607].ID := 1, [607].Active := 1, [608].ID := 2, [608].Active := 1, [609].ID := 1, [609].Active := 1, [610].ID := 2, [610].Active := 1, [611].ID := 1, [611].Active := 1, [612].ID := 2, [612].Active := 1, [613].ID := 1, [613].Active := 1, [614].ID := 2, [614].Active := 1, [615].ID := 1, [615].Active := 1, [616].ID := 2, [616].Active := 1, [617].ID := 1, [617].Active := 1, [618].ID := 2, [618].Active := 1, [619].ID := 1, [619].Active := 1, [620].ID := 2, [620].Active := 1, [621].ID := 1, [621].Active := 1, [622].ID := 2, [622].Active := 1, [623].ID := 1, [623].Active := 1, [624].ID := 2, [624].Active := 1, [625].ID := 1, [625].Active := 1, [626].ID := 2, [626].Active := 1, [627].ID := 1, [627].Active := 1, [628].ID := 2, [628].Active := 1, [629].ID := 1, [629].Active := 1,
        [630].ID := 2, [630].Active := 1, [631].ID := 1, [631].Active := 1, [632].ID := 2, [632].Active := 1, [633].ID := 1, [633].Active := 1, [634].ID := 2, [634].Active := 1, [635].ID := 1, [635].Active := 1, [636].ID := 2, [636].Active := 1, [637].ID := 1, [637].Active := 1, [638].ID := 2, [638].Active := 1, [639].ID := 1, [639].Active := 1, [640].ID := 2, [640].Active := 1, [641].ID := 1, [641].Active := 1, [642].ID := 2, [642].Active := 1, [643].ID := 1, [643].Active := 1, [644].ID := 2, [644].Active := 1, [645].ID := 1, [645].Active := 1, [646].ID := 2, [646].Active := 1, [647].ID := 1, [647].Active := 1, [648].ID := 2, [648].Active := 1, [649].ID := 1, [649].Active := 1, [650].ID := 2, [650].Active := 1, [651].ID := 1, [651].Active := 1, [652].ID := 2, [652].Active := 1, [653].ID := 1, [653].Active := 1, [654].ID := 2, [654].Active := 1, [655].ID := 1, [655].Active := 1, [656].ID := 2, [656].Active := 1, [657].ID := 1, [657].Active := 1, [658].ID := 2, [658].Active := 1, [659].ID := 1, [659].Active := 1,
        [660].ID := 2, [660].Active := 1, [661].ID := 1, [661].Active := 1, [662].ID := 2, [662].Active := 1, [663].ID := 1, [663].Active := 1, [664].ID := 2, [664].Active := 1, [665].ID := 1, [665].Active := 1, [666].ID := 2, [666].Active := 1, [667].ID := 1, [667].Active := 1, [668].ID := 2, [668].Active := 1, [669].ID := 1, [669].Active := 1, [670].ID := 2, [670].Active := 1, [671].ID := 1, [671].Active := 1, [672].ID := 2, [672].Active := 1, [673].ID := 1, [673].Active := 1, [674].ID := 2, [674].Active := 1, [675].ID := 1, [675].Active := 1, [676].ID := 2, [676].Active := 1, [677].ID := 1, [677].Active := 1, [678].ID := 2, [678].Active := 1, [679].ID := 1, [679].Active := 1, [680].ID := 2, [680].Active := 1, [681].ID := 1, [681].Active := 1, [682].ID := 2, [682].Active := 1, [683].ID := 1, [683].Active := 1, [684].ID := 2, [684].Active := 1, [685].ID := 1, [685].Active := 1, [686].ID := 2, [686].Active := 1, [687].ID := 1, [687].Active := 1, [688].ID := 2, [688].Active := 1, [689].ID := 1, [689].Active := 1,
        [690].ID := 2, [690].Active := 1, [691].ID := 1, [691].Active := 1, [692].ID := 2, [692].Active := 1, [693].ID := 1, [693].Active := 1, [694].ID := 2, [694].Active := 1, [695].ID := 1, [695].Active := 1, [696].ID := 2, [696].Active := 1, [697].ID := 1, [697].Active := 1, [698].ID := 2, [698].Active := 1, [699].ID := 1, [699].Active := 1, [700].ID := 2, [700].Active := 1, [701].ID := 1, [701].Active := 1, [702].ID := 2, [702].Active := 1, [703].ID := 1, [703].Active := 1, [704].ID := 2, [704].Active := 1, [705].ID := 1, [705].Active := 1, [706].ID := 2, [706].Active := 1, [707].ID := 1, [707].Active := 1, [708].ID := 2, [708].Active := 1, [709].ID := 1, [709].Active := 1, [710].ID := 2, [710].Active := 1, [711].ID := 1, [711].Active := 1, [712].ID := 2, [712].Active := 1, [713].ID := 1, [713].Active := 1, [714].ID := 2, [714].Active := 1, [715].ID := 1, [715].Active := 1, [716].ID := 2, [716].Active := 1, [717].ID := 1, [717].Active := 1, [718].ID := 2, [718].Active := 1, [719].ID := 1, [719].Active := 1,
        [720].ID := 2, [720].Active := 1, [721].ID := 1, [721].Active := 1, [722].ID := 2, [722].Active := 1, [723].ID := 1, [723].Active := 1, [724].ID := 2, [724].Active := 1, [725].ID := 1, [725].Active := 1, [726].ID := 2, [726].Active := 1, [727].ID := 1, [727].Active := 1, [728].ID := 2, [728].Active := 1, [729].ID := 1, [729].Active := 1, [730].ID := 2, [730].Active := 1, [731].ID := 1, [731].Active := 1, [732].ID := 2, [732].Active := 1, [733].ID := 1, [733].Active := 1, [734].ID := 2, [734].Active := 1, [735].ID := 1, [735].Active := 1, [736].ID := 2, [736].Active := 1, [737].ID := 1, [737].Active := 1, [738].ID := 2, [738].Active := 1, [739].ID := 1, [739].Active := 1, [740].ID := 2, [740].Active := 1, [741].ID := 1, [741].Active := 1, [742].ID := 2, [742].Active := 1, [743].ID := 1, [743].Active := 1, [744].ID := 2, [744].Active := 1, [745].ID := 1, [745].Active := 1, [746].ID := 2, [746].Active := 1, [747].ID := 1, [747].Active := 1, [748].ID := 2, [748].Active := 1, [749].ID := 1, [749].Active := 1,
        [750].ID := 2, [750].Active := 1, [751].ID := 1, [751].Active := 1, [752].ID := 2, [752].Active := 1, [753].ID := 1, [753].Active := 1, [754].ID := 2, [754].Active := 1, [755].ID := 1, [755].Active := 1, [756].ID := 2, [756].Active := 1, [757].ID := 1, [757].Active := 1, [758].ID := 2, [758].Active := 1, [759].ID := 1, [759].Active := 1, [760].ID := 2, [760].Active := 1, [761].ID := 1, [761].Active := 1, [762].ID := 2, [762].Active := 1, [763].ID := 1, [763].Active := 1, [764].ID := 2, [764].Active := 1, [765].ID := 1, [765].Active := 1, [766].ID := 2, [766].Active := 1, [767].ID := 1, [767].Active := 1, [768].ID := 2, [768].Active := 1, [769].ID := 1, [769].Active := 1, [770].ID := 2, [770].Active := 1, [771].ID := 1, [771].Active := 1, [772].ID := 2, [772].Active := 1, [773].ID := 1, [773].Active := 1, [774].ID := 2, [774].Active := 1, [775].ID := 1, [775].Active := 1, [776].ID := 2, [776].Active := 1, [777].ID := 1, [777].Active := 1, [778].ID := 2, [778].Active := 1, [779].ID := 1, [779].Active := 1,
        [780].ID := 2, [780].Active := 1, [781].ID := 1, [781].Active := 1, [782].ID := 2, [782].Active := 1, [783].ID := 1, [783].Active := 1, [784].ID := 2, [784].Active := 1, [785].ID := 1, [785].Active := 1, [786].ID := 2, [786].Active := 1, [787].ID := 1, [787].Active := 1, [788].ID := 2, [788].Active := 1, [789].ID := 1, [789].Active := 1, [790].ID := 2, [790].Active := 1, [791].ID := 1, [791].Active := 1, [792].ID := 2, [792].Active := 1, [793].ID := 1, [793].Active := 1, [794].ID := 2, [794].Active := 1, [795].ID := 1, [795].Active := 1, [796].ID := 2, [796].Active := 1, [797].ID := 1, [797].Active := 1, [798].ID := 2, [798].Active := 1, [799].ID := 1, [799].Active := 1, [800].ID := 2, [800].Active := 1, [801].ID := 1, [801].Active := 1, [802].ID := 2, [802].Active := 1, [803].ID := 1, [803].Active := 1, [804].ID := 2, [804].Active := 1, [805].ID := 1, [805].Active := 1, [806].ID := 2, [806].Active := 1, [807].ID := 1, [807].Active := 1, [808].ID := 2, [808].Active := 1, [809].ID := 1, [809].Active := 1,
        [810].ID := 2, [810].Active := 1, [811].ID := 1, [811].Active := 1, [812].ID := 2, [812].Active := 1, [813].ID := 1, [813].Active := 1, [814].ID := 2, [814].Active := 1, [815].ID := 1, [815].Active := 1, [816].ID := 2, [816].Active := 1, [817].ID := 1, [817].Active := 1, [818].ID := 2, [818].Active := 1, [819].ID := 1, [819].Active := 1, [820].ID := 2, [820].Active := 1, [821].ID := 1, [821].Active := 1, [822].ID := 2, [822].Active := 1, [823].ID := 1, [823].Active := 1, [824].ID := 2, [824].Active := 1, [825].ID := 1, [825].Active := 1, [826].ID := 2, [826].Active := 1, [827].ID := 1, [827].Active := 1, [828].ID := 2, [828].Active := 1, [829].ID := 1, [829].Active := 1, [830].ID := 2, [830].Active := 1, [831].ID := 1, [831].Active := 1, [832].ID := 2, [832].Active := 1, [833].ID := 1, [833].Active := 1, [834].ID := 2, [834].Active := 1, [835].ID := 1, [835].Active := 1, [836].ID := 2, [836].Active := 1, [837].ID := 1, [837].Active := 1, [838].ID := 2, [838].Active := 1, [839].ID := 1, [839].Active := 1,
        [840].ID := 2, [840].Active := 1, [841].ID := 1, [841].Active := 1, [842].ID := 2, [842].Active := 1, [843].ID := 1, [843].Active := 1, [844].ID := 2, [844].Active := 1, [845].ID := 1, [845].Active := 1, [846].ID := 2, [846].Active := 1, [847].ID := 1, [847].Active := 1, [848].ID := 2, [848].Active := 1, [849].ID := 1, [849].Active := 1, [850].ID := 2, [850].Active := 1, [851].ID := 1, [851].Active := 1, [852].ID := 2, [852].Active := 1, [853].ID := 1, [853].Active := 1, [854].ID := 2, [854].Active := 1, [855].ID := 1, [855].Active := 1, [856].ID := 2, [856].Active := 1, [857].ID := 1, [857].Active := 1, [858].ID := 2, [858].Active := 1, [859].ID := 1, [859].Active := 1, [860].ID := 2, [860].Active := 1, [861].ID := 1, [861].Active := 1, [862].ID := 2, [862].Active := 1, [863].ID := 1, [863].Active := 1, [864].ID := 2, [864].Active := 1, [865].ID := 1, [865].Active := 1, [866].ID := 2, [866].Active := 1, [867].ID := 1, [867].Active := 1, [868].ID := 2, [868].Active := 1, [869].ID := 1, [869].Active := 1,
        [870].ID := 2, [870].Active := 1, [871].ID := 1, [871].Active := 1, [872].ID := 2, [872].Active := 1, [873].ID := 1, [873].Active := 1, [874].ID := 2, [874].Active := 1, [875].ID := 1, [875].Active := 1, [876].ID := 2, [876].Active := 1, [877].ID := 1, [877].Active := 1, [878].ID := 2, [878].Active := 1, [879].ID := 1, [879].Active := 1, [880].ID := 2, [880].Active := 1, [881].ID := 1, [881].Active := 1, [882].ID := 2, [882].Active := 1, [883].ID := 1, [883].Active := 1, [884].ID := 2, [884].Active := 1, [885].ID := 1, [885].Active := 1, [886].ID := 2, [886].Active := 1, [887].ID := 1, [887].Active := 1, [888].ID := 2, [888].Active := 1, [889].ID := 1, [889].Active := 1, [890].ID := 2, [890].Active := 1, [891].ID := 1, [891].Active := 1, [892].ID := 2, [892].Active := 1, [893].ID := 1, [893].Active := 1, [894].ID := 2, [894].Active := 1, [895].ID := 1, [895].Active := 1, [896].ID := 2, [896].Active := 1, [897].ID := 1, [897].Active := 1, [898].ID := 2, [898].Active := 1, [899].ID := 1, [899].Active := 1,
        [900].ID := 2, [900].Active := 1, [901].ID := 1, [901].Active := 1, [902].ID := 2, [902].Active := 1, [903].ID := 1, [903].Active := 1, [904].ID := 2, [904].Active := 1, [905].ID := 1, [905].Active := 1, [906].ID := 2, [906].Active := 1, [907].ID := 1, [907].Active := 1, [908].ID := 2, [908].Active := 1, [909].ID := 1, [909].Active := 1, [910].ID := 2, [910].Active := 1, [911].ID := 1, [911].Active := 1, [912].ID := 2, [912].Active := 1, [913].ID := 1, [913].Active := 1, [914].ID := 2, [914].Active := 1, [915].ID := 1, [915].Active := 1, [916].ID := 2, [916].Active := 1, [917].ID := 1, [917].Active := 1, [918].ID := 2, [918].Active := 1, [919].ID := 1, [919].Active := 1, [920].ID := 2, [920].Active := 1, [921].ID := 1, [921].Active := 1, [922].ID := 2, [922].Active := 1, [923].ID := 1, [923].Active := 1, [924].ID := 2, [924].Active := 1, [925].ID := 1, [925].Active := 1, [926].ID := 2, [926].Active := 1, [927].ID := 1, [927].Active := 1, [928].ID := 2, [928].Active := 1, [929].ID := 1, [929].Active := 1,
        [930].ID := 2, [930].Active := 1, [931].ID := 1, [931].Active := 1, [932].ID := 2, [932].Active := 1, [933].ID := 1, [933].Active := 1, [934].ID := 2, [934].Active := 1, [935].ID := 1, [935].Active := 1, [936].ID := 2, [936].Active := 1, [937].ID := 1, [937].Active := 1, [938].ID := 2, [938].Active := 1, [939].ID := 1, [939].Active := 1, [940].ID := 2, [940].Active := 1, [941].ID := 1, [941].Active := 1, [942].ID := 2, [942].Active := 1, [943].ID := 1, [943].Active := 1, [944].ID := 2, [944].Active := 1, [945].ID := 1, [945].Active := 1, [946].ID := 2, [946].Active := 1, [947].ID := 1, [947].Active := 1, [948].ID := 2, [948].Active := 1, [949].ID := 1, [949].Active := 1, [950].ID := 2, [950].Active := 1, [951].ID := 1, [951].Active := 1, [952].ID := 2, [952].Active := 1, [953].ID := 1, [953].Active := 1, [954].ID := 2, [954].Active := 1, [955].ID := 1, [955].Active := 1, [956].ID := 2, [956].Active := 1, [957].ID := 1, [957].Active := 1, [958].ID := 2, [958].Active := 1, [959].ID := 1, [959].Active := 1,
        [960].ID := 2, [960].Active := 1, [961].ID := 1, [961].Active := 1, [962].ID := 2, [962].Active := 1, [963].ID := 1, [963].Active := 1, [964].ID := 2, [964].Active := 1, [965].ID := 1, [965].Active := 1, [966].ID := 2, [966].Active := 1, [967].ID := 1, [967].Active := 1, [968].ID := 2, [968].Active := 1, [969].ID := 1, [969].Active := 1, [970].ID := 2, [970].Active := 1, [971].ID := 1, [971].Active := 1, [972].ID := 2, [972].Active := 1, [973].ID := 1, [973].Active := 1, [974].ID := 2, [974].Active := 1, [975].ID := 1, [975].Active := 1, [976].ID := 2, [976].Active := 1, [977].ID := 1, [977].Active := 1, [978].ID := 2, [978].Active := 1, [979].ID := 1, [979].Active := 1, [980].ID := 2, [980].Active := 1, [981].ID := 1, [981].Active := 1, [982].ID := 2, [982].Active := 1, [983].ID := 1, [983].Active := 1, [984].ID := 2, [984].Active := 1, [985].ID := 1, [985].Active := 1, [986].ID := 2, [986].Active := 1, [987].ID := 1, [987].Active := 1, [988].ID := 2, [988].Active := 1, [989].ID := 1, [989].Active := 1,
        [990].ID := 2, [990].Active := 1, [991].ID := 1, [991].Active := 1, [992].ID := 2, [992].Active := 1, [993].ID := 1, [993].Active := 1, [994].ID := 2, [994].Active := 1, [995].ID := 1, [995].Active := 1, [996].ID := 2, [996].Active := 1, [997].ID := 1, [997].Active := 1, [998].ID := 2, [998].Active := 1);
   EVENT : CreatNewEvent := (Single_Input := 1, Ev_ID := 1);
   false : BOOL := 1;
   FSDF : TIME_To_STRING;
   io_Event : uEventsDB := (Events[0].ID := 1, Events[0].Active := 1, Events[0].Time.Yer := 1998, Events[0].Time.Month := 1, Events[0].Time.Day := 1, Events[0].Time.Hour := 5, Events[0].Time.Minute := 9, Events[0].Time.Sec := 48, Events[0].Time.MillSec := 396745, Events[1].ID := 1, Events[1].Active := 1, Events[1].Time.Yer := 2022, Events[1].Time.Month := 2, Events[1].Time.Day := 5, Events[1].Time.Hour := 14, Events[1].Time.Minute := 40, Events[1].Time.Sec := 40, Events[1].Time.MillSec := 175138, NextEvent := 1, RemainderValidEvent := 20);
   o_Err : BOOL;
   onshort : BOOL;
   S1 : BOOL := 1;
   Send_Event : CreateSendEvent;
   SSTR : STRING;
   Start : BOOL;
END_VAR

ROUTINE MainRoutine   (* ladder *)
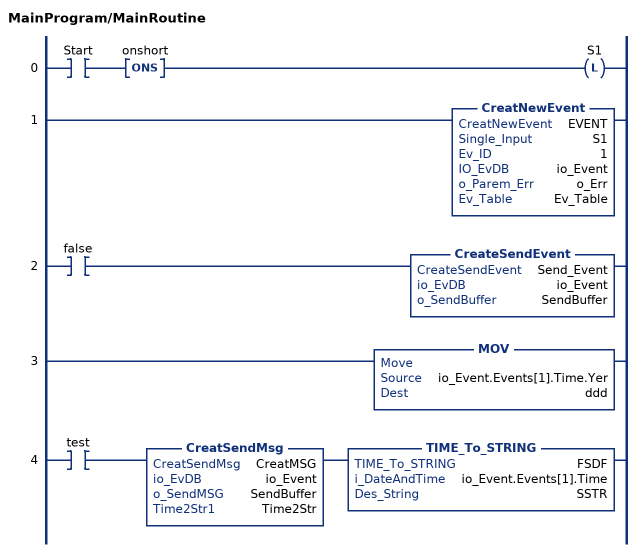
   0: XIC(Start)ONS(onshort)OTL(S1);
   1: CreatNewEvent(EVENT,S1,1,io_Event,o_Err,Ev_Table);
   2: XIC(false)CreateSendEvent(Send_Event,io_Event,SendBuffer);
   3: MOV(io_Event.Events[1].Time.Yer,ddd);
   4: XIC(test)CreatSendMsg(CreatMSG,io_Event,SendBuffer,Time2Str)TIME_To_STRING(FSDF,io_Event.Events[1].Time,SSTR);
END_ROUTINE
END_PROGRAM
